// TIA Portal V21 export
VAR_GLOBAL   // PLC tag table "K_QuoteMotoreAltezzaStampo"
END_VAR
VAR_GLOBAL CONSTANT   // user constants
   K_QuotaCarico : Int := 0;
   K_QuotaSteccatura : Int := 1;
   K_QuotaScarico : Int := 2;
END_VAR
